(*======================================================================================================================================*)
(*//=============================================================================\\
||  _   _ _  __  _         _                        _   _                      ||
|| | \ | | |/ / / \  _   _| |_ ___  _ __ ___   __ _| |_(_) ___  _ __         ||
|| |  \| | ' / / _ \| | | | __/ _ \| '_ ` _ \ / _` | __| |/ _ \| '_ \        ||
|| | |\  | . \/ ___ \ |_| | || (_) | | | | | | (_| | |_| | (_) | | | |       ||
|| |_| \_|_|\_\_/  \_\__,_|\__\___/|_| |_| |_|\__,_|\__|_|\___/|_| |_|       ||
||                                                                             ||
\\=============================================================================//
SERVOSCHRAUBER - Schraubprozess Schubkastenschiene Nobilia Vorgabe  

Dieser Baustein beschreibt den reinen Schraubprozess, es wird lediglich die 
Motoransteuerung übernommen, alles andere (Pneumatik und Schraubenzuführung) 
kann weiterhin in dem standart Schrauber Baustein stattfinden. Dies sorgt
für eine verbesserte Integration in bereits bestehende Systeme.

Die Gesamte Motoransteuerung findet über die "IQ_SchrauberAchsStruc_InOut" -
Achsstruktur statt, welche zusammen mit dem Baustein aufgerufen und beschrieben
wird. 

Über die "I_stSchraubParam" Struktur werden die Gesamten benötigten Parameter 
an den Schrauber- Baustein übergeben. Diese Struktur kann unverändert
durchgereicht werden.

================================================================================
Vollautomatischer Servoschrauber für Schienen- und Einzelschrauben
mit NC-Achsenanbindung, Drehmoment, Drehwinkel- und Tiefenüberwachung 
================================================================================*)

(*Date          | Version    		| created under     | Author       		| Remark *)
(*====================================================================================================================================================*)
(*23/09/2025   	| 1.00      		| TC3		  		| N.Kersting       	| Neue Isolierte Version *)
(*30/09/2025   	| 1.01      		| TC3		  		| N.Kersting       	| Erste Versuche ohne Motor  *)
(*01/10/2025   	| 1.02      		| TC3		  		| N.Kersting       	| Neue Strukturen Integriert für Prozessdaten etc. *)
(*08/10/2025   	| 1.03      		| TC3		  		| N.Kersting       	| Erste Versuche laufen sehr gut in der Praxis *)
(*09/10/2025   	| 1.04      		| TC3		  		| N.Kersting       	| Merhrere kleine Bugfixe/ Merker wurden nicht Initialisiert... *)
(*09/10/2025   	| 1.05      		| TC3		  		| N.Kersting       	| Drehmomenterhöhung in Schraubfall 1 und 3 nun über Zeit entprellt *)
(*09/10/2025   	| 2.00      		| TC3		  		| N.Kersting       	| Komplette Auswertungsstrategie abgespeckt und anderes konzept, ohne Tiefe zu beachten *)
(*10/10/2025   	| 3.00      		| TC3		  		| N.Kersting       	| Nach Drehmoment Ok wird nun auch die Schraubtiefe in Abhängikeit des Drehwinkels geprüft *)
(*10/10/2025   	| 3.01      		| TC3		  		| N.Kersting       	| Lauffähiger Stand, Auswertung sehr genau, Schraubzeit ca. 500-650ms *)
(*====================================================================================================================================================*)
FUNCTION_BLOCK fb_SKSSchraubNob
VAR_INPUT
	I_bStart			:BOOL;
	I_bFreigabe			:BOOL;
	I_bReset			:BOOL;
	I_bQuittFehler		:BOOL;
	
	I_lrActPosTiefe		:LREAL;
	
	I_stSchraubParam	:ST_SchrauberAblauf_Parameter;	(* Speziefische Parameter für den Schruabprozess *)
	
END_VAR
VAR_OUTPUT
	Q_sState			:STRING;
	Q_bBusy				:BOOL;
	Q_bDone				:BOOL;
	Q_bError			:BOOL;
	Q_nErrorId			:INT;
	Q_bSchrHalt			:BOOL;		(* Motor stoppen *)
	Q_bAxisReset		:BOOL;				(* Achse zurücksetzen *)
	Q_nTorque			:INT := 300;		(* Drehmomentgrenzwert [0.1%] *)
	
	Q_stProzessDaten	:ST_SchrauberAblauf_ProzessDaten;
END_VAR
VAR_IN_OUT
	(* Schraubantrieb Achsstruktur InOut *)
	IQ_SchrauberAchsStruc_InOut		:ST_SchrauberAblauf_AchsStruc;
END_VAR
VAR
	nStep				:INT;
	sStep				:STRING;
	nStepLeerlauf		:INT;
	sStepLeerlauf		:STRING;
	bBusy				: BOOL;
	bDone				: BOOL;
	
	(*========================================================================================================================*)
	(* === PROZESSWERTE === *)
	(*========================================================================================================================*)
	fSchraubTiefeIst				: LREAL;	(* Aktuelle Schraubtiefe [mm] *)
	fDrehmomentIstMittel			: LREAL;	(* Gemitteltes Drehmoment [0.1%] *)
	nTiefeBeimAufsetzen				: LREAL;	(* Tiefe beim ersten Werkstückkontakt *)
	bTiefeBeimAufsetzenOK			: BOOL;		(* Aufsetzen korrekt erkannt *)
	bTiefeOkMem						: BOOL;
	bDrehmomOkMem					: BOOL;
	bDrehwinkelOkMem				: BOOL;
	bTiefeStehtOkMem				: BOOL;
	bSchraubStangeStehtOkMem		: BOOL;
	bDrehwinkelTiefeOkMem			: BOOL;
	nDrehwinkelMem					: LREAL ;
	nTiefErrechnetMem				: LREAL;
	nTiefeAbweichMem				: LREAL;
	nSollDrehmomentErrechnet		: LREAL;	(* Der errechnete Drehmomentwert, Rechnet Drehmoment (Nm) um in Prozessdaten kompatibelen wert für den Antrieb! *)
	bLeerlaufpruefung				: BOOL;
	bDrehmomentErhoehen				: BOOL;			(* Merker Drehmoment erhöhen *)
	bAchsreset						: BOOL;		(* Achsen-Reset intern *)
	lrDrehzahlSollProzent			: LREAL;
	
	(*========================================================================================================================*)
	(* === FEHLERBEHANDLUNG === *)
	(*========================================================================================================================*)
	nFehlerSchrittMerker			: INT;		(* Merker für Fehlerschritt *)
	
	(*========================================================================================================================*)
	(* === Prozessparameter zur Schraubfall auswertung === *)
	(*========================================================================================================================*)
	nAuswertungTiefeMem				: LREAL;	(* Gemerkte Tiefe für Auswertung in Step 60 *)
	nAuswertungPosMem				: LREAL;	(* Gemerkte Position für Auswertung in Step 60 *)
	nMaxDrehwinkel_F3				: LREAL;			
	nDrehwinkelBerechnet			: LREAL; 			(* Der Maximale solldrehwinkel, welcher sich aus der Höhe, wo gestoppt wurde und der Schraubensteigung errechnet *)
	nSchraubFallMerker				: INT;	
	nDrehmomentSkalierVorgabe		: LREAL;
	
	(*========================================================================================================================*)
	(* === Auswertung === *)
	(*========================================================================================================================*)
	fbtimeDiff_Schraub				: fb_timeDiff;
	fbtimeDiff_Komplettt			: fb_timeDiff;
	rTrigPosMem						: r_trig;
	
	(*========================================================================================================================*)
	(* === Zeiten === *)
	(*========================================================================================================================*)
	tonTimeOver						: ton;
	tonDrehmomentErhoehen			: ton;
	
	(*========================================================================================================================*)
	(* === DREHMOMENT-MITTELWERTBILDUNG === *)
	(*========================================================================================================================*)
	arrDrehmomentIst				: ARRAY [0..10] OF LREAL;	(* Ringpuffer für Drehmoment *)
	idx								: INT;		(* Index für Array-Verarbeitung *)
	
	(*========================================================================================================================*)
	(* === Prozesswerte für Analyse === *)
	(*========================================================================================================================*)
	nPD_Tiefe						: LREAL;			(* Prozessdaten - erreichte Tiefe *)
	nPD_Drehmoment					: LREAL;			(* Prozessdaten - erreichtes Drehmoment *)
	nPD_Drehwinkel					: LREAL;			(* Prozessdaten - erreichter Drehwinkel *)
	tPD_Schraubtakt_Komplett		: TIME;				(* Prozessdaten - Zeit für den Kompletten Schraubprozess *)
	tPD_Schraubtakt_Schrauben		: TIME;				(* Prozessdaten - Zeit nur für den Schraubvorgang ohne Zylinder bewegungen etc. *)
	iPD_Schraubfall					: INT;				(* Prozessdaten - Schraubfall *)		
	bPD_SchraubVorgOk				: BOOL;				(* Prozessdaten - Schraubvorgang OK *)
	
	nSollDrehzahl					: INT;
	
	fbtimeDiff_Step45				: fb_timeDiff;
	fbtimeDiff_Step50				: fb_timeDiff;
	fbtimeDiff_Step51				: fb_timeDiff;
	fbtimeDiff_Step55				: fb_timeDiff;
	fbtimeDiff_Step60				: fb_timeDiff;
	fbtimeDiff_Step61				: fb_timeDiff;
	fbtimeDiff_Step62				: fb_timeDiff;
	fbtimeDiff_Step70				: fb_timeDiff;
	fbtimeDiff_Step75				: fb_timeDiff;
	
	stArraySteps					: ARRAY[1..9] OF STRING;
	tGesamtZeit						: TIME;
	sGesamtZeit						: STRING;
	i								: INT;
	rTrigZeitenSchreiben			: R_trig;
	
END_VAR

fSchraubTiefeIst :=	I_lrActPosTiefe;

(* === Hauptablauf === *)
ac_Hauptablauf();

(* === DREHMOMENT-MITTELWERTBILDUNG === *)
m_DrehmomentMittelwert();

(* === SCHRAUBTAKT-ZEITMESSUNG === *)
m_SchraubtaktMessung();

(* === Ausgänge zuweisen === *)
m_Ausgangszuweisung();

ACTION ac_AblaufLeerlaufPruef:
(* ================================================================================ *)
(* LERRLAUF DREHMOMENT PRÜFEN SEQUENZ *)
(* ================================================================================ *)
CASE nStepLeerlauf OF
0: (* === LeerlaufPrüfung/ Erkennung ob Motor Schwergängig ist === *)
	sStepLeerlauf := 'Leerlaufpruefung';
			
	(* Watchdog Positionierfreigabe *)
	tonTimeOver.IN := TRUE;
	tonTimeOver.PT := T#1S;
		
	(* Startdrehzahl setzen *)
	m_DrehzahlVorgabe(
		lrMaxDrehzahl:=  		IQ_SchrauberAchsStruc_InOut.NC_Axis_IN_nParamEilgeschw, 
		lrDrehzahlSollUpm:= 	I_stSchraubParam.nDrehzahlSollEnde, 
		lrDrehzahlVorgabe=> 	lrDrehzahlSollProzent);
			
	(* Drehmoment Vorgabe errechnen *)
	m_DrehmomentVorgabe(
		nSkalierung :=			1,
		nTorque:= 				I_stSchraubParam.nSollmomentLeerlaufPruefung, (* Lerrlaufdrehmoment *) 
		nRatedCurrentMotor:= 	I_stSchraubParam.nNennleistungMotor, 
		nTorqueConstant:= 		I_stSchraubParam.nDrehmomentKonstante, 
		nTorqueLimitation=> 	nSollDrehmomentErrechnet);
		
	Q_nTorque := LREAL_TO_INT(nSollDrehmomentErrechnet);
	
	IF IQ_SchrauberAchsStruc_InOut.NC_Axis_IN_bPTPPosiFreig
	THEN
		tonTimeOver.IN := FALSE;
		
		IQ_SchrauberAchsStruc_InOut.NC_Axis_OUT_nPTPVelo := lrDrehzahlSollProzent;
		IQ_SchrauberAchsStruc_InOut.NC_Axis_OUT_PTPBuffMode := MC_Aborting;
		IQ_SchrauberAchsStruc_InOut.NC_Axis_OUT_bAchsePosStarten := TRUE;	
		nStepLeerlauf := 301;
	ELSIF
		tonTimeOver.Q
	THEN
		tonTimeOver.IN := FALSE;
		nFehlerSchrittMerker := -300;
		nStepLeerlauf := 999;
	END_IF
	
(*================================================================================================================*)
1: (* === LeerlaufPrüfung === *)
	sStepLeerlauf := 'Leerlaufpruefung Auswertung';
	
	(* Watchdog für Leerlauf Prüfung ob Geschwindigkeit mit reduziertem Drehmoment erreicht wurde *)
	(* Watchdog Positionierfreigabe *)
	tonTimeOver.IN := IQ_SchrauberAchsStruc_InOut.NC_Axis_IN_bFaehrtPos;(* Muss noch geguckt werden ob auchh bei Stillstehendem Motor gesetzt wird *)
	tonTimeOver.PT := I_stSchraubParam.tLeerlaufPruefzeit;(* warten damit die Drehzahl erreicht werden kann *)
	
	bLeerlaufpruefung := TRUE;

	(* Wenn 80% der Solldrehzahl erreicht wurde, gilt dies als OK *)
	IF  (((IQ_SchrauberAchsStruc_InOut.NC_Axis_IN_nActVelo / IQ_SchrauberAchsStruc_InOut.NC_Axis_IN_nParamEilgeschw) * 100)
		 >= IQ_SchrauberAchsStruc_InOut.NC_Axis_OUT_nPTPVelo*0.8)
	THEN
		tonTimeOver.IN := FALSE;
		nStepLeerlauf := 999;
	ELSIF
		tonTimeOver.Q
	THEN
		tonTimeOver.IN := FALSE;
		nFehlerSchrittMerker := -301;
		nStepLeerlauf := 999;
	END_IF	

999:;
	
END_CASE
END_ACTION

ACTION ac_Hauptablauf:
(*
================================================================================
HAUPTABLAUF - ZUSTANDSMASCHINE SERVOSCHRAUBER
================================================================================
Zentrale Zustandsmaschine mit deterministischem Ablauf.
Alle Schritte sind eindeutig nummeriert und kommentiert.
Watchdog-Timer überwachen kritische Phasen.
================================================================================
*)

tonTimeOver();

(*=== HAUPTZUSTANDSMASCHINE === *)
IF NOT I_bReset 
THEN
	CASE nStep OF
(*================================================================================================================*)	
	(* ================================================================================ *)
	(* INITIALISIERUNG UND BEREITSCHAFT *)
	(* ================================================================================ *)
(*================================================================================================================*)
	0: (* === INITIALISIERUNG === *)
		sStep := 'Initialisierung';
		bDone := FALSE;
		
		(* Drehmoment Vorgabe errechnen *)
		m_DrehmomentVorgabe(
			nSkalierung :=			I_stSchraubParam.nDrehmomentSkalierVorgabe,
			nTorque:= 				I_stSchraubParam.nDrehmomentSoll * I_stSchraubParam.nDrehmomentSkalierVorgabe, (* Drehmoment erst Senken um Überdrehen zu verhinder *) 
			nRatedCurrentMotor:= 	I_stSchraubParam.nNennleistungMotor, 
			nTorqueConstant:= 		I_stSchraubParam.nDrehmomentKonstante, 
			nTorqueLimitation=> 	nSollDrehmomentErrechnet);
			
		Q_nTorque := LREAL_TO_INT(nSollDrehmomentErrechnet); 
		
		IF I_bFreigabe
		THEN
			nStep := 10;
		END_IF
		
(*================================================================================================================*)
	10: (* === BEREITSCHAFT === *)
		sStep := 'Bereitschaft';
		tonTimeOver.IN := FALSE;
		tonDrehmomentErhoehen.IN := FALSE;
		
		(* Drehmoment Vorgabe errechnen *)
		m_DrehmomentVorgabe(
			nSkalierung :=			I_stSchraubParam.nDrehmomentSkalierVorgabe,
			nTorque:= 				I_stSchraubParam.nDrehmomentSoll * I_stSchraubParam.nDrehmomentSkalierVorgabe, (* Drehmoment erst Senken um Überdrehen zu verhinder *) 
			nRatedCurrentMotor:= 	I_stSchraubParam.nNennleistungMotor, 
			nTorqueConstant:= 		I_stSchraubParam.nDrehmomentKonstante, 
			nTorqueLimitation=> 	nSollDrehmomentErrechnet);
			
		Q_nTorque := LREAL_TO_INT(nSollDrehmomentErrechnet); 
		bBusy							:= TRUE;
		
		IF I_bStart
			AND Q_nTorque <>0
		THEN
			(* Prozessdaten auf 0 setzen *)
			nPD_Tiefe						:= 0;			(* Prozessdaten - erreichte Tiefe *)
			nPD_Drehmoment					:= 0;			(* Prozessdaten - erreichtes Drehmoment *)
			nPD_Drehwinkel					:= 0;			(* Prozessdaten - erreichter Drehwinkel *)
			tPD_Schraubtakt_Komplett		:= T#0S;		(* Prozessdaten - Zeit für den Kompletten Schraubprozess *)
			tPD_Schraubtakt_Schrauben		:= T#0S;		(* Prozessdaten - Zeit nur für den Schraubvorgang ohne Zylinder bewegungen etc. *)
			iPD_Schraubfall					:= 0;			(* Prozessdaten - Schraubfall *)		
			bPD_SchraubVorgOk				:= FALSE;		(* Prozessdaten - Schraubvorgang OK *)
			nDrehwinkelMem     				:= 0;
			bDrehmomOkMem					:= FALSE;
			bDrehwinkelOkMem				:= FALSE;
			bTiefeOkMem						:= FALSE;
			bTiefeStehtOkMem				:= FALSE;
			bDrehmomentErhoehen				:= FALSE;
			bSchraubStangeStehtOkMem		:= FALSE;
			bDrehwinkelTiefeOkMem			:= FALSE;
			nTiefeAbweichMem				:= 0;
			nFehlerSchrittMerker			:= 0;
			nSchraubFallMerker				:= 0;
			nTiefErrechnetMem				:= 0;
			nStep := 45;
		END_IF
		
(*================================================================================================================*)
	45: (* === ANLAUFPHASE - LANGSAME DREHZAHL === *)
		sStep := 'Anlaufphase_Langsam';
					
		(* Watchdog für Anlaufphase *)
		tonTimeOver.IN := TRUE;
		tonTimeOver.PT := T#5S;
	
		(* Startdrehzahl setzen *)
		m_DrehzahlVorgabe(
			lrMaxDrehzahl:=  		IQ_SchrauberAchsStruc_InOut.NC_Axis_IN_nParamEilgeschw, 
			lrDrehzahlSollUpm:= 	I_stSchraubParam.nDrehzahlSollAnfang, 
			lrDrehzahlVorgabe=> 	lrDrehzahlSollProzent);
			
		IQ_SchrauberAchsStruc_InOut.NC_Axis_OUT_nPTPVelo := lrDrehzahlSollProzent;
		IQ_SchrauberAchsStruc_InOut.NC_Axis_OUT_PTPBuffMode := MC_Aborting;
		IQ_SchrauberAchsStruc_InOut.NC_Axis_OUT_bAchsePosStarten := I_bFreigabe;
		
		(* Prüfung ob 80% der Sollgeschwindigkeit erreicht *)
		IF	IQ_SchrauberAchsStruc_InOut.NC_Axis_IN_bFaehrtPos 
		    AND (((IQ_SchrauberAchsStruc_InOut.NC_Axis_IN_nActVelo / IQ_SchrauberAchsStruc_InOut.NC_Axis_IN_nParamEilgeschw) * 100)
			     >= IQ_SchrauberAchsStruc_InOut.NC_Axis_OUT_nPTPVelo * 0.8)
		THEN
			
			IQ_SchrauberAchsStruc_InOut.NC_Axis_OUT_bAchsePosStarten := FALSE;
			tonTimeOver.IN := FALSE;
			nStep := 50;	(* -> Hauptschraubphase *)
			
		ELSIF tonTimeOver.Q 
		THEN
			(* Timeout - Geschwindigkeit nicht erreicht *)
			tonTimeOver.IN := FALSE;
			nStep := 70;	(* -> Motor stoppen *)
			nFehlerSchrittMerker := -45;	(* Fehlercode merken *)
		END_IF
		
(*================================================================================================================*)
	50: (* === HAUPTSCHRAUBPHASE - GESCHWINDIGKEIT AUFBAUEN === *)
		sStep := 'Hauptschraubphase_Beschleunigen';
		
		(* Watchdog für Beschleunigungsphase *)
		tonTimeOver.IN := TRUE;
		tonTimeOver.PT := T#3S;
			
		IQ_SchrauberAchsStruc_InOut.NC_Axis_OUT_bAchsePosStarten := I_bFreigabe;
		
		(* Prozessdaten Tiefe Schreiben *)
		nPD_Tiefe:=	fSchraubTiefeIst;
		
		(* Startdrehzahl setzen *)
		m_DrehzahlVorgabe(
			lrMaxDrehzahl:=  		IQ_SchrauberAchsStruc_InOut.NC_Axis_IN_nParamEilgeschw, 
			lrDrehzahlSollUpm:= 	I_stSchraubParam.nDrehzahlSoll, 
			lrDrehzahlVorgabe=> 	lrDrehzahlSollProzent);
			
		(* Umschaltung auf Solldrehzahl basierend auf Schraubtiefe *)
		IF I_bStart 
			AND fSchraubTiefeIst < I_stSchraubParam.nTiefeSollDrehzahl 
		THEN
			(* Vollschraubung *)
			tonTimeOver.IN := FALSE;
			IQ_SchrauberAchsStruc_InOut.NC_Axis_OUT_bAchsePosStarten := FALSE;
			IQ_SchrauberAchsStruc_InOut.NC_Axis_OUT_nPTPVelo := lrDrehzahlSollProzent;
			IQ_SchrauberAchsStruc_InOut.NC_Axis_OUT_PTPBuffMode := MC_BlendingNext;
			IQ_SchrauberAchsStruc_InOut.NC_Axis_OUT_bAchsePosStarten := I_bFreigabe;
			nStep := 51;	(* -> Drehzahlabsenkung *)
		ELSIF 
			tonTimeOver.Q 
		THEN
			(* Timeout - Solltiefe für Drehzahlumschaltung nicht erreicht *)
			tonTimeOver.IN := FALSE;
			nStep := 70;	(* -> Motor stoppen *)
			nFehlerSchrittMerker := -50;	(* Fehlercode merken *)
		END_IF
		
(*================================================================================================================*)
	51: (* === Warten Auf Velo Verringert === *)
		sStep := 'Hauptschraubphase_Drehzahl verringern';	
		
		(* Watchdog für Beschleunigungsphase *)
		tonTimeOver.IN := TRUE;
		tonTimeOver.PT := I_stSchraubParam.tZeitdSchraubTakt;
			
		(* Startdrehzahl setzen *)
		m_DrehzahlVorgabe(
			lrMaxDrehzahl:=  		IQ_SchrauberAchsStruc_InOut.NC_Axis_IN_nParamEilgeschw, 
			lrDrehzahlSollUpm:= 	I_stSchraubParam.nDrehzahlSollEnde, 
			lrDrehzahlVorgabe=> 	lrDrehzahlSollProzent);
		
		(* Aufruf Drehmoment Prüfen *)
		m_DrehmomentPruefung(
			nDrehmomentSoll:= 		I_stSchraubParam.nDrehmomentSoll, 
			bDrehmomentOk=> 		bDrehmomOkMem);
	
		IF fSchraubTiefeIst < I_stSchraubParam.nTiefeLangsamDrehzahl
			OR bDrehmomOkMem	(* Nun auch schon vorher gucken ob das Drehmoment nicht doch schon kommt um Drehzahl zu Reduzieren *)
		THEN
			(* Vollschraubung *)
			IQ_SchrauberAchsStruc_InOut.NC_Axis_OUT_bAchsePosStarten := I_bFreigabe;
			IQ_SchrauberAchsStruc_InOut.NC_Axis_OUT_nPTPVelo := lrDrehzahlSollProzent  ;	
			IQ_SchrauberAchsStruc_InOut.NC_Axis_OUT_PTPBuffMode := MC_BlendingNext;
			IQ_SchrauberAchsStruc_InOut.NC_Axis_OUT_bAchsePosStarten := I_bFreigabe;
		
			(* Warten, dass 80% der iSt Drehzahl kleiner ist als die Soll Drehzahl  *)
			IF IQ_SchrauberAchsStruc_InOut.NC_Axis_IN_bFaehrtPos 
				AND (((IQ_SchrauberAchsStruc_InOut.NC_Axis_IN_nActVelo*0.8 / IQ_SchrauberAchsStruc_InOut.NC_Axis_IN_nParamEilgeschw) * 100)
					 <= IQ_SchrauberAchsStruc_InOut.NC_Axis_OUT_nPTPVelo)	
			THEN
				tonTimeOver.IN := FALSE;
				nStep := 55;	
			END_IF
			
		ELSIF
			tonTimeOver.Q
		THEN			
			tonTimeOver.IN := FALSE;
			nFehlerSchrittMerker := -51;	(* -> Timeout Kein Drehmoment und keine Tiefe *) (* Fehlercode merken *)
			nStep := 70;	
		END_IF
		
(*================================================================================================================*)
	55: (* === Schraubfallauswertung === *)
		sStep := 'Schraubfall Auswertung';
		
		(* Watchdog für Auswertung Schraubfall *)
		tonTimeOver.IN := TRUE;
		tonTimeOver.PT := I_stSchraubParam.tSchraubfallAuswertung;
			
		IQ_SchrauberAchsStruc_InOut.NC_Axis_OUT_bAchsePosStarten := I_bFreigabe;
		
		(* Startdrehzahl setzen *)
		m_DrehzahlVorgabe(
			lrMaxDrehzahl:=  		IQ_SchrauberAchsStruc_InOut.NC_Axis_IN_nParamEilgeschw, 
			lrDrehzahlSollUpm:= 	I_stSchraubParam.nDrehzahlSollEnde, 
			lrDrehzahlVorgabe=> 	lrDrehzahlSollProzent);
		
		(* Tiefenprüfung *)
		IF I_bStart
		THEN
			m_TiefenPruefung(
				nSolltiefeMin:= 	I_stSchraubParam.nMinimalSchraubtiefe, 
				nSolltiefeMax:= 	I_stSchraubParam.nSchraubtiefeSoll, 
				nToleranz:= 		0,	 
				nActTiefe:= 		fSchraubTiefeIst, 
				bTiefeOk=> 			bTiefeOkMem);
		END_IF
		
		(* Aufruf Drehmoment Prüfen *)
		m_DrehmomentPruefung(
			nDrehmomentSoll:= 		I_stSchraubParam.nDrehmomentSoll, 
			bDrehmomentOk=> 		bDrehmomOkMem);
					
		IF bDrehmomOkMem
		THEN
			tonTimeOver.IN := FALSE;
			IQ_SchrauberAchsStruc_InOut.NC_Axis_OUT_nPTPVelo := lrDrehzahlSollProzent ;	
			nSchraubFallMerker :=	1;
			nStep := 60;
		ELSIF
			 tonTimeOver.Q 
		THEN							
			tonTimeOver.IN := FALSE;
			nFehlerSchrittMerker := -55;	(* -> Timeout Drehmoment erreichen *) (* Fehlercode merken *)
			nStep := 70;	
		END_IF
		
(*================================================================================================================*)
	60: (* === Warten Auf Velo Verringert === *)
		sStep := 'Schraubfall Auswertung';	
		
		(* Watchdog für Schraubvorgang *)
		tonTimeOver.IN := TRUE;
		tonTimeOver.PT :=  I_stSchraubParam.tZeitdSchraubTakt;
		
		(* Warten, dass 80% der iSt Drehzahl kleiner ist als die Soll Drehzahl  *)
		IF IQ_SchrauberAchsStruc_InOut.NC_Axis_IN_bFaehrtPos 
		    AND (((IQ_SchrauberAchsStruc_InOut.NC_Axis_IN_nActVelo*0.8 / IQ_SchrauberAchsStruc_InOut.NC_Axis_IN_nParamEilgeschw) * 100)
			     <= IQ_SchrauberAchsStruc_InOut.NC_Axis_OUT_nPTPVelo)
		THEN
			nAuswertungPosMem := IQ_SchrauberAchsStruc_InOut.NC_Axis_IN_nActPos; (* Position Merken, wo Drehmoment erreicht wurde *)	
			nAuswertungTiefeMem :=	fSchraubTiefeIst; (* Tiefe Merken, wo Drehmoment erreicht wurde *)
					
			nStep := 61;	
		ELSIF
			tonTimeOver.Q
		THEN			
			tonTimeOver.IN := FALSE;
			nFehlerSchrittMerker := -60;	(* -> Timeout Drehzahl Absenken *) (* Fehlercode merken *)
			nStep := 70;	
		END_IF
		
(*================================================================================================================*)			
	61:	(* === Schraubfall === *) 
		ac_Schraubfall();	
		
(*================================================================================================================*)			
	62:	(* === Tiefenänderung prüfen === *) 
		ac_TiefenAuswertung();
		
(*================================================================================================================*)			
(*	63:	(* === Schraubfall 3 === *) 
		ac_Schraubfall3();		*)
		
(*================================================================================================================*)
	70: (* === MOTOR STOPPEN === *)
		sStep := 'Motor_Stoppen';
		Q_nTorque := 0;
		
		(* Watchdog für Stoppvorgang *)
		tonTimeOver.IN := TRUE;
		tonTimeOver.PT :=  T#100MS;
				
		(* Achse stoppen *)
		IQ_SchrauberAchsStruc_InOut.NC_Axis_OUT_bAchsePosStoppen := TRUE;
		
		(* Warten auf Stillstand *)
		IF tonTimeOver.Q 
		   OR IQ_SchrauberAchsStruc_InOut.NC_Axis_IN_bInPos
		THEN
			tonTimeOver.IN := FALSE;
			IQ_SchrauberAchsStruc_InOut.NC_Axis_OUT_bAchsePosStoppen := FALSE;
			IQ_SchrauberAchsStruc_InOut.NC_Axis_OUT_bAchsePosStarten := FALSE;
			nStep := 75;	(* -> Stillstand abwarten *)
		END_IF
		
(*================================================================================================================*)
	75: (* === STILLSTAND ABWARTEN === *)
		sStep := 'Stillstand_Abwarten';
		
		(* Watchdog für Stillstand *)
		tonTimeOver.IN := TRUE;
		tonTimeOver.PT :=  T#2S;
		
		(* Warten auf Motorstillstand *)
		IF tonTimeOver.Q
			OR IQ_SchrauberAchsStruc_InOut.NC_Axis_IN_bInStillstand
		THEN
			bAchsreset := TRUE;
			tonTimeOver.IN := FALSE;
			
			nStep := 80;
		END_IF

(*================================================================================================================*)
	80: (* === AUSWERTUNG FEHLERSCHRITTMERKER === *)
		sStep := 'Fehlerschritt auswerten';
		
		(* Fehler auswerten *)
		IF nFehlerSchrittMerker <> 0
		THEN
			nStep := nFehlerSchrittMerker;
		ELSE
			bPD_SchraubVorgOk := TRUE;
			nStep := 100;
		END_IF
				
(*================================================================================================================*)
	100: (* === VORGANG ERFOLGREICH BEENDET === *)
		sStep := 'Vorgang_OK';
		
		bBusy := FALSE;
		bDone := TRUE;
		
		(* Warten auf Freigabe für nächsten Zyklus *)
		IF NOT I_bStart 
		THEN
			bLeerlaufpruefung := FALSE;
			Q_nTorque := 300;	
			IQ_SchrauberAchsStruc_InOut.NC_Axis_OUT_bSteuerwortBit1	:= FALSE;
			IQ_SchrauberAchsStruc_InOut.NC_Axis_OUT_bAchsePosStarten := FALSE;
			nStep := 0;	(* -> Zurück zur Bereitschaft *)
		END_IF
		
(*================================================================================================================*)
	(* ================================================================================ *)
	(* LERRLAUF DREHMOMENT PRÜFEN SEQUENZ *)
	(* ================================================================================ *)
	300: sStep := sStepLeerlauf;
				
		ac_AblaufLeerlaufPruef();
		
		IF nStepLeerlauf = 999
		THEN
			nStepLeerlauf :=0;
			nStep := 70;
		END_IF
		
(*================================================================================================================*)
	(* ================================================================================ *)
	(* FEHLERBEHANDLUNG *)
	(* ================================================================================ *)
		
(*================================================================================================================*)
	-45: (* === FEHLER: LANGSAME GESCHWINDIGKEIT === *)
		sStep := 'FEHLER: Langsame Geschwindigkeit wird nicht erreicht';
		Q_nErrorId := -45;
		
		IF I_bQuittFehler 
		THEN
			nStep := 100;	(* -> Beenden *)
		END_IF
		
(*================================================================================================================*)
	-50: (* === FEHLER: SCHRAUBTIEFE FÜR SOLLDREHZAHL === *)
		sStep := 'FEHLER: Schraubtiefe für Solldrehzahl wird nicht erreicht';
		Q_nErrorId := -50;
		
		IF I_bQuittFehler 
		THEN
			nStep := 100;	(* -> Beenden *)
		END_IF
		
(*================================================================================================================*)
	-55: (* === FEHLER:  === *)
		sStep := 'FEHLER: Timeout Drehmoment- Auswertung';
		Q_nErrorId := -55;
		
		IF I_bQuittFehler 
		THEN
			nStep := 100;	(* -> Beenden *)
		END_IF
		
(*================================================================================================================*)		
	-60: (* === FEHLER:  === *)
		sStep := 'FEHLER: Timeout abbremsen';
		Q_nErrorId := -60;
		
		IF I_bQuittFehler 
		THEN
			nStep := 100;	(* -> Beenden *)
		END_IF
		
(*================================================================================================================*)
(* === FEHLER: Schraubfall 1  === *)		
(*================================================================================================================*)
	-61: 
		sStep := 'FEHLER: Schraubfall 1 Undefiniert- Timeout';
		Q_nErrorId := -61;
		
		IF I_bQuittFehler 
		THEN
			nStep := 100;	(* -> Beenden *)
		END_IF
		
(*================================================================================================================*)
	-1261: 
		sStep := 'FEHLER: Schraubfall 1 Drehwinkel Überschritten';
		Q_nErrorId := -1261;
		
		IF I_bQuittFehler 
		THEN
			nStep := 100;	(* -> Beenden *)
		END_IF	
		
(*================================================================================================================*)
	-62: 
		sStep := 'FEHLER: Tiefe hat sich geändert obwohl Drehmoment OK';
		Q_nErrorId := -62;
		
		IF I_bQuittFehler 
		THEN
			nStep := 100;	(* -> Beenden *)
		END_IF
		
(*================================================================================================================*)
	-301: (* === FEHLER: Leerlaufprüfung === *)
		sStep := 'FEHLER: Leerlauf Drehzahl nicht erreicht, Schwergang?';
		Q_nErrorId := -301;
		
		IF I_bQuittFehler 
		THEN
			nStep := 100;	(* -> Beenden *)
		END_IF
		
(*================================================================================================================*)
	-300: (* === FEHLER: Leerlaufprüfung === *)
		sStep := 'FEHLER: Leerlaufprüfung keine Freigabe zum Positionieren';
		Q_nErrorId := -300;
		
		IF I_bQuittFehler 
		THEN
			nStep := 100;	(* -> Beenden *)
		END_IF
		
	END_CASE
	
ELSE
	(* === RESET AKTIV === *)
	nStep := 0;
END_IF

(*========================================================*)
(* Prozessdaten Merker schreiben *)
(*========================================================*)
IF (nStep >= 55)
	AND (nStep <= 70)
THEN
	(* Prozessdaten Drehwinkel Schreiben *)
	IF nDrehwinkelMem> nPD_Drehwinkel
	THEN
		nPD_Drehwinkel :=	nDrehwinkelMem;
	END_IF
	(* Prozessdaten Tiefe Schreiben *)
	IF fSchraubTiefeIst < nPD_Tiefe
	THEN
		nPD_Tiefe:=	fSchraubTiefeIst;
	END_IF
	(* Prozessdaten Drehmoment Schreiben *)
	IF fDrehmomentIstMittel >nPD_Drehmoment
	THEN
		nPD_Drehmoment :=	fDrehmomentIstMittel;
	END_IF
	
	iPD_Schraubfall :=	nSchraubFallMerker;
END_IF

(*========================================================*)
(* Prozessdaten Struktur schreiben *)
(*========================================================*)
Q_stProzessDaten.nPD_Drehmoment				:=	nPD_Drehmoment;
Q_stProzessDaten.nPD_Drehwinkel				:=	nPD_Drehwinkel;
Q_stProzessDaten.nPD_Tiefe					:=	nPD_Tiefe;
Q_stProzessDaten.tPD_Schraubtakt_Komplett	:=	tPD_Schraubtakt_Komplett;
Q_stProzessDaten.tPD_Schraubtakt_Schrauben	:=	tPD_Schraubtakt_Schrauben;
Q_stProzessDaten.iPD_Schraubfall			:=	iPD_Schraubfall;
Q_stProzessDaten.bPD_SchraubVorgOk			:=	bPD_SchraubVorgOk;
Q_stProzessDaten.bPD_DrehmomOk				:=	bDrehmomOkMem;
Q_stProzessDaten.bPD_DrehwinkelOk			:=	bDrehwinkelOkMem;
Q_stProzessDaten.bPD_TiefeOk				:=	bTiefeOkMem;
END_ACTION

ACTION ac_Schraubfall:
(*================================================================================================================*)
(* === Drehwinkelprüfung&  Drehmoment Prüfung === *)
(*
Fall 1 – Moment OK, Tiefe nicht OK
- Ausgangslage: Verbindung zieht, Tiefe fehlt noch.
- Ziel: Tiefer eindrehen, ohne Überdrehen.
- Vorgehen:
  - Weiterdrehen mit großer Winkelreserve.
  - Reserve aus fehlender Tiefe + Schraubensteigung berechnet,
    plus kleiner Nachziehwinkel.
- Stop: Tiefe erreicht innerhalb Reserve → Stopp.
- Eskalation: Tiefe kommt nicht → Moment moderat erhöhen.
- Abbruch: Timeout oder Winkelobergrenze überschritten.*)
(*================================================================================================================*)

sStep := 'Schraubvorgang Auswertung Drehwinkel und Drehmoment';

(* Watchdog für Schraubvorgang *)
tonTimeOver.IN := 	TRUE;
tonTimeOver.PT :=	I_stSchraubParam.tZeitdSchraubfallTimeout;

Q_nTorque := LREAL_TO_INT(nSollDrehmomentErrechnet );	(* Drehmoment wieder Setzen damit der Motor weiter drehen kann *)

(* Aufruf Drehwinkel Prüfen *)
m_DrehwinkelPruefung(
	nPosAct:= 			IQ_SchrauberAchsStruc_InOut.NC_Axis_IN_nActPos, 
	nPosMem:= 			nAuswertungPosMem, 
	nPosSoll:= 			I_stSchraubParam.nSollDrehwinkelNachDrehmomOK, (* mindest Drehwinkel nach Drehmoment ok *)
	nMaxDrehwinkel :=	I_stSchraubParam.nMaxDrehwinkelNachDrehmOk, (* Maximal Drehwinkel nach Drehmoment ok *)
	bWinkelOk=> 		bDrehwinkelOkMem,
	nWinkelAct=>		nDrehwinkelMem);

(* Aufruf Drehmoment Prüfen *)
m_DrehmomentPruefung(
	nDrehmomentSoll:= 		I_stSchraubParam.nDrehmomentSoll, 
	bDrehmomentOk=> 		bDrehmomOkMem);

(* Aufruf Schrauberstange auf Stillstand Prüfen *)	
m_StillstandPruef(
	nIstDrehzahl:= 		IQ_SchrauberAchsStruc_InOut.NC_Axis_IN_nActVelo, 
	nMinDrehzahl:= 		ABS(IQ_SchrauberAchsStruc_InOut.NC_Axis_IN_nParamEilgeschw * 0.01), (* 1% der Bezugsgeschwindigkeit *)
	bSteht=> 			bSchraubStangeStehtOkMem);
	
IF NOT tonTimeOver.Q
THEN
	IF 	ABS(nDrehwinkelMem) <I_stSchraubParam.nMaxDrehwinkelNachDrehmOk	(* Nur abfragen ob nicht überdreht *)
		AND bSchraubStangeStehtOkMem (* Schrauberstange dreht sich nicht mehr *) 
		AND bDrehmomOkMem
	THEN 	
		tonTimeOver.IN := 	FALSE;
		Q_nTorque := 0;
		nStep := 62;	(* -> Motor stoppen *)
	ELSIF
		ABS(nDrehwinkelMem) >(I_stSchraubParam.nMaxDrehwinkelNachDrehmOk)
	THEN
		(* Wenn Drehwinkel Überschritten-> Direkt Anhalten *)
		tonTimeOver.IN := 	FALSE;
		nStep := 70;	(* -> Motor stoppen *)
		nFehlerSchrittMerker := -1261;	(* Fehlercode merken Drehwinkel Überschritten Fall 1*)			
	END_IF
ELSE
	nFehlerSchrittMerker := -61;
	tonTimeOver.IN := 	FALSE;
	nStep := 70;	(* -> Motor stoppen *)
END_IF
END_ACTION

ACTION ac_TiefenAuswertung:
(* Watchdog für Tiefenänderung *)
tonTimeOver.IN := TRUE;
tonTimeOver.PT :=  T#100MS;

m_TiefenAenderung(
	nTiefeStreckeIst:= 		ABS(fSchraubTiefeIst) -ABS(nAuswertungTiefeMem), 
	nDrehwinkelIst:= 		nDrehwinkelMem, 
	nSteigungSchraube:= 	I_stSchraubParam.nHoeheSchraubenDrehung, 
	nAbweichung:= 			25, 
	nTiefeErrechnet=> 		nTiefErrechnetMem, 
	nProzentAbweichung=>	nTiefeAbweichMem,
	bTiefeSteht=> 			bTiefeStehtOkMem);
 
IF bTiefeStehtOkMem
THEN
	tonTimeOver.IN := 	FALSE;
	Q_nTorque := 0;
	nStep := 70;	(* -> Motor stoppen *)
ELSIF
	tonTimeOver.Q
THEN
	(* Wenn bTiefeStehtOkMem bedeutet dies, dass der Schraubenkopf noch nicht anliegt, 
		weiterer Umgang muss noch Folgen, aber erst mal Fehler*)
	tonTimeOver.IN := FALSE;
	nFehlerSchrittMerker := -62;	(* -> Tiefe hat sich geändert Logik muss noch folgen, aber erst mal Fehler *) (* Fehlercode merken *)
	nStep := 70;
END_IF
END_ACTION

ACTION ac99_Doku:
(*
## 1. Überblick / Zweck
Der Baustein `fb_SKSSchraubNob` kapselt den **reinen servo‑motorischen Schraubprozess** (Drehzahl-, Drehmoment-, Winkel- und Tiefenführung) und lässt alle peripheren Funktionen (z. B. Pneumatik, Schraubenzuführung) im bestehenden Standard-Schrauberbaustein. Dadurch kann der Motor-Schraubkern in bestehende Anlagen integriert werden, ohne tiefgreifende Umbauten in der Peripherie vornehmen zu müssen.  
Unterstützt werden:
- Drehmomentüberwachung  
- Drehwinkelberechnung / -begrenzung  
- Tiefenerfassung (Position entspricht Einschraubtiefe)  
- Klassifizierung des Verlaufs in definierte Schraubfälle  
- Zeit- und Qualitätsauswertung  

## 2. Integration in einen vorhandenen Schrauberablauf
Einbettung erfolgt typischerweise so:
1. Bestehender Ablauf (PnP / Handlingslogik) positioniert Werkzeug, versorgt Schraube, setzt ggf. Pneumatik.
2. Achsstruktur (IN/OUT) wird an den Baustein übergeben (standardisierte Servoantriebs-Schnittstelle).
3. Parametrierstruktur (Schraubparameter) wird 1:1 durchgereicht (keine Aufsplittung nötig).
4. Start-/Freigabe-/Reset-/Quittiersignale kommen aus übergeordneter Ablaufsteuerung.
5. Prozessdaten (Tiefe, Drehmoment, Winkel, Dauer, Klassifikation) werden nach Abschluss zurückgemeldet und können für Trace, Qualität oder MES erfasst werden.
6. Fehler- oder Schraubfall-Ergebnis kann direkt in nachfolgende Entscheider (OK/NOK/Sortierung) einfließen.

Vorteile:
- Plug-in für bestehenden Schrauber-Ablauf .
- Leichte Austauschbarkeit oder parallele Variantenentwicklung.
- Geringeres Risiko bei Änderungen (nur Kernlogik betroffen).
- Einheitliche Achsschnittstelle fördert Wiederverwendung.

## 3. Architektur & Zustandslogik (technischer Überblick)
Der Baustein verwendet eine deterministische Zustandsmaschine (nummerierte Schritte). Kernphasen:
1. Initialisierung / Bereitschaft
2. Anlauf mit reduzierter Drehzahl
3. Übergang auf Hauptdrehzahl
4. Drehzahlreduktion vor Auswertung
5. Schraubfall-Erkennung (Entscheidung: welcher Verlauf liegt vor?)
6. Feinschraubphase je nach Schraubfall (1, 2 oder 3)
7. Bremsen / Stillsetzen
8. Ergebnis- und Fehlerauswertung
9. Rückkehr in Bereitschaft

Ergänzend: eigene Sequenz zur Leerlauf-/Schwergangprüfung mit separater Unter-Zustandsmaschine.

## 4. Schraubfälle (Klassifikation des Verlaufs)
Die Klassifikation beruht auf der Relation zwischen erreichten Zielgrößen (Tiefe, Drehmoment) zum Zeitpunkt der Auswertung:

| Schraubfall | Auslöser (Situation) | Zielstrategie | Typische Maßnahmen | Abbruchkriterien |
|-------------|----------------------|---------------|--------------------|------------------|
| 1 | Drehmoment erreicht, Tiefe noch nicht | Weiter eindringen ohne Überdrehen | Winkelreserve aus fehlender Tiefe + Nachziehreserve, ggf. Drehmoment moderat erhöhen | Timeout, Winkelgrenze überschritten |
| 2 | Tiefe erreicht, Drehmoment noch nicht | Vorspannung sauber aufbauen | Begrenztes Nachdrehen in kleinem Winkel-Fenster | Timeout (Moment fehlt), Fenster überschritten |
| 3 | Weder Tiefe noch Moment erreicht | Beides sicher erreichen | Zunächst größere Winkel-/Tiefenreserve, dann Übergang wie Fall 1 bzw. 2 | Timeout, Winkelobergrenze |
| Leerlaufprüfung | Vor dem eigentlichen Prozess: Antrieb läuft „frei“ | Erkennen von Schwergang / Blockade | Prüfen ob Geschwindigkeit mit reduziertem Moment erreicht wird | Timeout oder zu niedrige Drehzahl |

Zusammenfassung:
- Fall 1: Verbindung zieht früh (Moment da), Schraube steht noch sichtbar über Oberfläche.
- Fall 2: Schraube liegt bündig (Tiefe da), aber Vorspannung fehlt noch.
- Fall 3: „Träger Verlauf“ – weder Tiefe noch Moment früh erreicht, daher weiter beobachten und adaptiv reagieren.
- Leerlaufprüfung: Schutzmechanismus / Frühdiagnose.

## 5. Ablaufbeschreibung 
1. Der Baustein wartet, bis die übergeordnete Steuerung signalisiert, dass alles bereit ist (Werkzeug positioniert, Schraube vorhanden, Sicherheitsfreigaben aktiv).
2. Beim Start setzt er interne Messgrößen (z. B. Zähler und Qualitätsmerker) zurück.
3. Der Schraubvorgang beginnt langsam, um ein ruckfreies Ansetzen sicherzustellen und frühe Auffälligkeiten (Blockade, verkantete Schraube) zu erkennen.
4. Erhöht sich die Einschraubtiefe wie erwartet, wird beschleunigt, um Zeit zu sparen.
5. Kurz vor einer vorgesehenen Übergangszone wird wieder auf eine niedrigere Geschwindigkeit reduziert, um kontrolliert in den sensiblen Bereich (Finalisierung) einzufahren.
6. Nun vergleicht das System: Ist bereits die benötigte Tiefe erreicht? Ist das gewünschte Drehmoment erzielt? Aus dieser Kombination erkennt es, welcher Verlauf vorliegt.
7. Je nach Verlauf wendet es ein passendes Feinkonzept an:
   - Schraubfall 1: Nur Tiefe fehlt → etwas weiter eindrehen, ohne zu fest anzuziehen.
   - Schraubfall 2: Nur Drehmoment fehlt → gezielte Nachdrehung, begrenzt im Winkel.
   - Schraubfall 3: Beides fehlt → weitere kontrollierte Bewegung, mit eventueller Anpassung.
8. Währenddessen wird laufend das Drehmoment gemittelt um Ausreißer zu filtern.
9. Erreichen alle Zielgrößen gültige Werte (Tiefe im Fenster, Drehmoment ausreichend, Winkel nicht zu groß), wird der Antrieb gestoppt.
10. Der Prozess wird protokolliert: Zeitbedarf, erreichte Tiefe, maximales Drehmoment, gedrehter Winkel und Klassifikation.
11. Bei Unregelmäßigkeiten (z. B. Zeit überschritten, Winkel zu groß) markiert das System den Vorgang als fehlerhaft und wartet auf eine Quittierung.
12. Nach Freigabe für den nächsten Zyklus kehrt der Baustein in die Ausgangsbereitschaft zurück.


## 6. Prozessdaten (Ergebnis- / Qualitätsdaten)
| Name (Ausgabe) | Bedeutung | Einheit | Hinweise |
|----------------|----------|---------|----------|
| nPD_Tiefe | Erreichte minimale Einschraubtiefe (negativer Weg oder mm je nach Bezug) | mm | Wird während der aktiven Phase aktualisiert (kleinster Wert, falls Tiefe Richtung Werkstück negativ zählt) |
| nPD_Drehmoment | Höchstes gemitteltes Drehmoment im Prozess | % (0.1%-Skalierung) oder intern skaliert | Basierend auf Mittelwertbildung zur Glättung |
| nPD_Drehwinkel | Größter errechneter/erfasster Drehwinkel (Differenz seit Auswertungspunkt) | Grad / Umdrehungsäquivalent | Berechnet aus Achsposition und Steigung |
| tPD_Schraubtakt_Komplett | Gesamtzeit von Start bis Abschluss/Fehler | Zeit | Für Taktoptimierung |
| tPD_Schraubtakt_Schrauben | Reine Schraubzeit (ohne z. B. Zylinderwege) | Zeit | Differenziert Ursachen von Verzögerungen |
| iPD_Schraubfall | Klassifizierter Schraubfall (1–3) | Zahl | 0 vor Auswertung |
| bPD_SchraubVorgOk | Gesamt-OK-Flag des Vorgangs | BOOL | FALSE bei Fehler oder Abbruch |
| bPD_DrehmomOk | Soll-Drehmoment erreicht | BOOL | Teilkriterium Qualität |
| bPD_DrehwinkelOk | Nachdreh-/Winkelkriterium erfüllt | BOOL | Verhindert Überdrehen |
| bPD_TiefeOk | Tiefe innerhalb Toleranzfenster | BOOL | Oberflächenbündigkeit / Setzpunkt |

## 7. Parameterbeschreibung (Eingabestruktur)
(Hinweis: Nicht alle Parameter der Struktur waren vollständig sichtbar. Liste basiert auf den im Code referenzierten Feldern.)

| Parameter | Bedeutung / Funktion | Einheit / Bereich | Wirkung / Bemerkungen |
|-----------|----------------------|-------------------|-----------------------|
| nDrehzahlSollAnfang | Anfangsdrehzahl für Schon-Anlauf | U/min | Reduziert Risiko von Verkanten |
| nDrehzahlSoll | Hauptdrehzahl (Schnellphase) | U/min | Produktivgeschwindigkeit |
| nDrehzahlSollEnde | Reduzierte Drehzahl in Feinschraubphase | U/min | Feinfühliges Erreichen der Ziele |
| nTiefeSollDrehzahl | Einschraubtiefe, ab der auf Hauptdrehzahl hochgeschaltet wird | mm | Umschaltkriterium Beschleunigung |
| nTiefeLangsamDrehzahl | Einschraubtiefe, ab der wieder verlangsamt wird | mm | Vorbereitung Feinauswertung |
| nMinimalSchraubtiefe | Untere Toleranzgrenze für Tiefe | mm | Qualitätsfenster |
| nSchraubtiefeSoll | Zieltiefe | mm | Nennwert Tiefe |
| nDrehmomentSoll | Ziel-Drehmoment | Skaliert / % / Nm-Äquivalent | Referenz für Freigabekriterium |
| nDrehmomentSkalierVorgabe | Globaler Skalierungsfaktor | Faktor | Multipliziert Ziel-Moment (z. B. Softstart) |
| nDrehmomentSkalVerringern | Temporäre Reduktion für Brems-/Übergangsphase | Faktor | Vor Auswertung wird Moment gesenkt |
| nDrehmomentErhoehung | Zusatzmoment bei Fall 1 / 3 wenn Tiefe „hängt“ | Skaliert | Adaptive Nachregelung |
| nSollmomentLeerlaufPruefung | Momentbegrenzung in Leerlaufprüfung | % / skaliert | Erkennung Schwergang ohne Schäden |
| tLeerlaufPruefzeit | Prüfzeitfenster Leerlauf | Zeit | Timeout-Kriterium |
| tZeitdSchraubTakt | Allgemeines Zeitlimit für Teilphasen / Nachziehfenster | Zeit | Wiederverwendetes Watchdog-Intervall |
| tSchraubfallAuswertung | Spezifisches Zeitfenster für Klassifikation | Zeit | Verhindert endloses Abwarten |
| nHoeheSchraubenDrehung | Steigung (Tiefe pro Umdrehung oder pro Segment) | mm/U | Grundlage für Winkelberechnung |
| nSollDrehwinkelNachTiefeOK | Mindestnachdrehwinkel nach Tiefeerfüllung | Grad | Sicherstellung Setzvorgang |
| nDrehwinkelNachziehen_F1 | Zusatz-Winkelreserve bei Fall 1 | Grad | Verhindert Untervorspannung |
| nMaxDrehwinkelNachTiefeOk_F1 | Sicherheitslimit Fall 1 | Grad | Abbruch bei Überdrehung |
| nMaxDrehwinkelNachTiefeOk_F2 | Sicherheitslimit Fall 2 | Grad | Engeres Fenster |
| (vermutet) nMaxDrehwinkel_F3 | Limit für Fall 3 (im Code angelegt) | Grad | Analog Fall 1/2 (nicht komplett sichtbar) |
| nNennleistungMotor | Referenz Motorstrom / Bemessung | A / % | Für Berechnung Drehmomentgrenze |
| nDrehmomentKonstante | Umrechnungsfaktor (Strom→Moment) | Nm/A | Erforderlich für physikalische Skalierung |
*)
END_ACTION

METHOD m_Ausgangszuweisung : BOOL
VAR_INPUT
END_VAR
(*
================================================================================
AUSGANGSZUWEISUNG
================================================================================
Zentrale Zuweisung aller Ausgangssignale mit Sicherheitsverriegelung
durch Schutzbereich und Reset-Zustand
================================================================================
*)

// === HAUPTSTATUS-AUSGÄNGE ===
Q_bBusy		:= bBusy;				(* Beschäftigt wenn nicht in Bereitschaft *)

Q_bDone		:= bDone;		(* Fertig bei Schritt 100 *)

// === ACHSEN-STEUERUNG ===
Q_bAxisReset := bAchsreset;

// === DIAGNOSE-AUSGÄNGE ===
Q_sState	:= sStep(*CONCAT(INT_TO_STRING(nStep), CONCAT(' - ', sStep))*);

Q_bSchrHalt := (nStep = 70);

(* Fehler allgemein *)
Q_bError	:= nStep<0;
END_METHOD

METHOD m_DrehmomentMittelwert : BOOL
VAR_INPUT
END_VAR
(*
================================================================================
DREHMOMENT-MITTELWERTBILDUNG
================================================================================
Berechnet den gleitenden Mittelwert des Drehmoments über 10 Werte
zur Vermeidung von Fehlauslösungen durch kurze Spitzen.
================================================================================
*)
// === MITTELWERTBILDUNG NUR WÄHREND DREHMOMENTPRÜFUNG ===
IF (nStep >= 51 
	AND nStep <= 70) 
	OR nStep =301
THEN
	m_DrehmomentRechnung(
		nTorqueActValue:= 		INT_TO_LREAL(IQ_SchrauberAchsStruc_InOut.NC_Axis_IN_nActTorque), 
		nRatedCurrentMotor:=	I_stSchraubParam.nNennleistungMotor , 	
		nTorqueConstant:= 		I_stSchraubParam.nDrehmomentKonstante, 
		nActTorqueCalc=> 		arrDrehmomentIst[0]);
	
	// Array nach rechts verschieben (Ringpuffer)
	FOR idx := 10 TO 1 BY -1 DO
		arrDrehmomentIst[idx] := arrDrehmomentIst[idx-1];
	END_FOR
	
	// Mittelwert über alle 10 Werte berechnen
	fDrehmomentIstMittel := (arrDrehmomentIst[1] 
						   + arrDrehmomentIst[2] 
						   + arrDrehmomentIst[3] 
						   + arrDrehmomentIst[4] 
						   + arrDrehmomentIst[5] 
						   + arrDrehmomentIst[6] 
						   + arrDrehmomentIst[7] 
						   + arrDrehmomentIst[8] 
						   + arrDrehmomentIst[9] 
						   + arrDrehmomentIst[10]) / 10;
ELSE
	fDrehmomentIstMittel := 0;
END_IF
END_METHOD

METHOD m_DrehmomentPruefung : BOOL
VAR_INPUT
	nDrehmomentSoll		:LREAL;				
END_VAR
VAR_OUTPUT
	bDrehmomentOk		:BOOL;
END_VAR
(*
================================================================================
DrehmomentPruefung
================================================================================
Berechnet den gleitenden Mittelwert des Drehmoments über 10 Werte
zur Vermeidung von Fehlauslösungen durch kurze Spitzen.
================================================================================
*)
IF fDrehmomentIstMittel >= 
	nDrehmomentSoll
THEN
	bDrehmomentOk := TRUE;	(* -> Drehmoment erreicht *)
ELSE
	bDrehmomentOk := FALSE;	
END_IF
END_METHOD

METHOD m_DrehmomentRechnung : BOOL
VAR_INPUT
	
	
	nTorqueActValue		:LREAL;	
	
	nRatedCurrentMotor	:LREAL;	(*0x8011:12	*)
	nTorqueConstant		:LREAL;	(*0x8011:16	*)
END_VAR
VAR_OUTPUT
	nActTorqueCalc		:LREAL;
END_VAR
(*Achtung dies aus der Original Beckhoff Doku:

Anzeige des aktuellen Drehmomentwertes
Der Wert wird in 1000stel vom rated current (0x8011:12
[} 151]) angegeben
Formel für Index 0x8010:54 [} 148] = 0 :
M = ((Torque actual value / 1000) x (rated current /
√2)) x torque constant (0x8011:16 [} 151])
Formel für Index 0x8010:54 [} 148] = 1 :
M = ((Torque actual value / 1000) x rated current)) x
torque constant (0x8011:16 [} 151])*)
nActTorqueCalc:=	
(((nTorqueActValue/1000) * (nRatedCurrentMotor / 1.4142))* nTorqueConstant);		(* Wurzel ziehen am besten einmalig bei Startup *)
END_METHOD

METHOD m_DrehmomentVorgabe : BOOL
VAR_INPUT
	nSkalierung			:LREAL;
	nTorque				:LREAL;		(* Eingang Soll Drehmoment in Nm	*)
	
	nRatedCurrentMotor	:LREAL;	(*0x8011:12	*)
	nTorqueConstant		:LREAL;	(*0x8011:16	*)
END_VAR
VAR_OUTPUT
	nTorqueLimitation	:LREAL;
END_VAR
(*Achtung dies aus der Original Beckhoff Doku:

Anzeige des aktuellen Drehmomentwertes
Der Wert wird in 1000stel vom rated current (0x8011:12
[} 151]) angegeben
Formel für Index 0x8010:54 [} 148] = 0 :
M = ((Torque actual value / 1000) x (rated current /
√2)) x torque constant (0x8011:16 [} 151])
Formel für Index 0x8010:54 [} 148] = 1 :
M = ((Torque actual value / 1000) x rated current)) x
torque constant (0x8011:16 [} 151])*)
nTorqueLimitation := ((nTorque / nTorqueConstant) / (nRatedCurrentMotor / 1.4142)) * 1000 *nSkalierung;
END_METHOD

METHOD m_DrehwinkelPruefung : BOOL
VAR_INPUT
	nPosAct		:LREAL;	(* Aktuelle Position  *)
	nPosMem		:LREAL;	(* Gespeicherte Position *)
	nPosSoll	:LREAL; (* Soll Drehwinkel *)
	nMaxDrehwinkel	:LREAL;
	
END_VAR
VAR_OUTPUT
	bWinkelOk			:BOOL;
	nWinkelAct	:LREAL;
END_VAR
VAR
	
END_VAR
nWinkelAct :=	nPosAct-nPosMem;

bWinkelOk :=	nWinkelAct > nPosSoll 
				AND nWinkelAct < nMaxDrehwinkel;
END_METHOD

METHOD m_DrehzahlVorgabe 
VAR_INPUT
	lrMaxDrehzahl		:LREAL;		(* Drhezahl Eilgeschwindigkeit in Grad/ sec *)
	lrDrehzahlSollUpm	:LREAL;		(* Drehzahl Soll in Upm *)
END_VAR
VAR
	lrDrehzahlMem		:LREAL;
	
END_VAR
VAR_OUTPUT
	lrDrehzahlVorgabe	:LREAL;			(* Soll Drehzahl in % von 100 % *)
END_VAR
lrDrehzahlMem := lrMaxDrehzahl /360 *60;

IF lrDrehzahlMem <> 0
THEN
	lrDrehzahlVorgabe :=	lrDrehzahlSollUpm / lrDrehzahlMem *100;
END_IF
END_METHOD

METHOD m_SchraubtaktMessung : BOOL
VAR_INPUT
END_VAR
(*
================================================================================
SCHRAUBTAKT-ZEITMESSUNG
================================================================================
Misst die Schraubzeit für Diagnose und Optimierung.
Die Zeitmessung erfolgt während der aktiven Schraubphase.
================================================================================
*)
(* Komplett wird nicht verwendet, da ausgelagert in dem Übergeordneten Schrauberbaustein *)
(*fbtimeDiff_Komplettt(
	bStart:= 		(nStep =10),	 
	bStop:= 		(nStep =100), 
	bReset:= 		(nStep =10),
	tDiffTime=> 	tPD_Schraubtakt_Komplett);*)
	
tPD_Schraubtakt_Komplett := T#0MS;

(* Zeitmessung Schruabvorgang *)
fbtimeDiff_Schraub(
	bStart:= 		(nStep =45),	 
	bStop:= 		(nStep =80), 
	bReset:= 		(nStep =10),
	tDiffTime=> 	tPD_Schraubtakt_Schrauben);

	
fbtimeDiff_Step45(
	bStart:= 			nStep =45, 
	bStop:= 			nStep <>45, 
	bReset:= 			nStep = 10);

fbtimeDiff_Step50(
	bStart:= 			nStep =50, 
	bStop:= 			nStep <>50, 
	bReset:= 			nStep = 10);
	
fbtimeDiff_Step51(
	bStart:= 			nStep =51, 
	bStop:= 			nStep <>51, 
	bReset:= 			nStep = 10);
	
fbtimeDiff_Step55(
	bStart:= 			nStep =55, 
	bStop:= 			nStep <>55, 
	bReset:= 			nStep = 10);
	
fbtimeDiff_Step60(
	bStart:= 			nStep =60, 
	bStop:= 			nStep <>60, 
	bReset:= 			nStep = 10);
	
fbtimeDiff_Step45(
	bStart:= 			nStep =45, 
	bStop:= 			nStep <>45, 
	bReset:= 			nStep = 10);
	
fbtimeDiff_Step61(
	bStart:= 			nStep =61, 
	bStop:= 			nStep <>61, 
	bReset:= 			nStep = 10);
	
fbtimeDiff_Step62(
	bStart:= 			nStep =62, 
	bStop:= 			nStep <>62, 
	bReset:= 			nStep = 10);

fbtimeDiff_Step70(
	bStart:= 			nStep =70, 
	bStop:= 			nStep <>70, 
	bReset:= 			nStep = 10);

fbtimeDiff_Step75(
	bStart:= 			nStep =75, 
	bStop:= 			nStep <>75, 
	bReset:= 			nStep = 10);	
	
(* Zeiten Schreiben *)
rTrigZeitenSchreiben(CLK:= (nStep =100));

IF rTrigZeitenSchreiben.Q
THEN
	stArraySteps[1] :=	CONCAT('Step_45_LangsamEin: ', INT_TO_STRING(TIME_TO_INT(fbtimeDiff_Step45.tDiffTime )));
	stArraySteps[2] :=	CONCAT('Step_50_Beschleunigen auf SollDrehzahl: ', INT_TO_STRING(TIME_TO_INT(fbtimeDiff_Step50.tDiffTime )));
	stArraySteps[3] :=	CONCAT('Step_51_Umschaltung Langsame Drehzahl: ', INT_TO_STRING(TIME_TO_INT(fbtimeDiff_Step51.tDiffTime )));
	stArraySteps[4] :=	CONCAT('Step_55_Warte auf Drehmoment: ', INT_TO_STRING(TIME_TO_INT(fbtimeDiff_Step55.tDiffTime )));
	stArraySteps[5] :=	CONCAT('Step_60_Warte auf Drehzahl verringert: ', INT_TO_STRING(TIME_TO_INT(fbtimeDiff_Step60.tDiffTime )));
	stArraySteps[6] :=	CONCAT('Step_61_Auswertung Drehmoment und Drehwinkel: ', INT_TO_STRING(TIME_TO_INT(fbtimeDiff_Step61.tDiffTime )));
	stArraySteps[7] :=	CONCAT('Step_62_Auswertung Tiefenänderung: ', INT_TO_STRING(TIME_TO_INT(fbtimeDiff_Step62.tDiffTime )));
	stArraySteps[8] :=	CONCAT('Step_70_Motor anhalten: ', INT_TO_STRING(TIME_TO_INT(fbtimeDiff_Step70.tDiffTime )));
	stArraySteps[9] :=	CONCAT('Step_75_Warte auf Motor Steht: ', INT_TO_STRING(TIME_TO_INT(fbtimeDiff_Step75.tDiffTime )));
	
	tGesamtZeit:=	fbtimeDiff_Step45.tDiffTime
					+	fbtimeDiff_Step50.tDiffTime
					+	fbtimeDiff_Step51.tDiffTime
					+	fbtimeDiff_Step55.tDiffTime
					+	fbtimeDiff_Step60.tDiffTime
					+	fbtimeDiff_Step61.tDiffTime
					+	fbtimeDiff_Step62.tDiffTime
					+	fbtimeDiff_Step70.tDiffTime
					+	fbtimeDiff_Step75.tDiffTime;
					
	sGesamtZeit :=		CONCAT('GesamtZeit: ', INT_TO_STRING(TIME_TO_INT(tGesamtZeit )));
END_IF
END_METHOD

METHOD m_StillstandPruef 
VAR_INPUT
	nIstDrehzahl	:LREAL;
	nMinDrehzahl	:LREAL;
END_VAR
VAR_OUTPUT
	bSteht			:BOOL;
END_VAR




IF ABS(nIstDrehzahl) < ABS(nMinDrehzahl) 
THEN
	bSteht := TRUE;
ELSE
	bSteht := FALSE;
END_IF
END_METHOD

METHOD m_TiefenAenderung
VAR_INPUT
	nTiefeStreckeIst				:LREAL;
	nDrehwinkelIst					:LREAL;
	nSteigungSchraube				:LREAL := 1.6;	(* Tiefe pro umdrehung *)
	nAbweichung						:LREAL := 25;	(* in Prozent *)
END_VAR
VAR_OUTPUT
	nProzentAbweichung 				:LREAL;	(* Nur zu Diagnosezwecken *)
	nTiefeErrechnet					:LREAL;	(* Nur zu Diagnosezwecken *)
	bTiefeSteht						:BOOL;
END_VAR
VAR
	nDelta             : LREAL;
END_VAR

IF nSteigungSchraube  > 0
	AND nAbweichung > 0
THEN
	nTiefeErrechnet :=	ABS(nDrehwinkelIst /360* nSteigungSchraube);
	
	nDelta := ABS(nTiefeErrechnet - nTiefeStreckeIst);
	
    IF nTiefeStreckeIst <> 0.0 THEN
        nProzentAbweichung := nDelta / ABS(nTiefeStreckeIst) * 100.0;
    ELSE
        nProzentAbweichung := 0.0;
    END_IF

    IF nProzentAbweichung >= nAbweichung THEN
        bTiefeSteht := TRUE;
    ELSE
        bTiefeSteht := FALSE;
    END_IF
	
ELSE
    bTiefeSteht := FALSE;
    nTiefeErrechnet := 0.0;
END_IF
END_METHOD

METHOD m_TiefenPruefung : BOOL
VAR_INPUT
	nSolltiefeMin	:LREAL;
	nSolltiefeMax	:LREAL;
	nToleranz	:LREAL;
	nActTiefe	:LREAL;
END_VAR
VAR_OUTPUT
	bTiefeOk	:BOOL;
END_VAR
// Prüfung der Aufsetztiefe
IF F_Inbetween(
	I_fActualValue := nActTiefe,
	I_fMinimalValue := nSolltiefeMin - nToleranz,		(* Sollaufsetztiefe ± Toleranz *)
	I_fMaximalValue := nSolltiefeMax + nToleranz) 
THEN
	bTiefeOk := TRUE;
ELSE
	bTiefeOk := FALSE;
END_IF
END_METHOD

END_FUNCTION_BLOCK

(* stored: Version 1.1.0.1, ProductVersion 3.1.4024.15
   POU fb_SKSSchraubNob: Id {7264520c-c401-4547-9877-f980c7765746}, SpecialFunc None
   Folder Ablauf: Id {fafa4d6d-6f22-46f3-bf08-cf1d510a3348}
   Folder Ausgang: Id {6aba5681-4e5c-480a-99f0-c6a63017ffef}
   Folder Auswertung: Id {6546e813-580a-4c40-8d8a-37f1e1c6b5fe}
   Folder Diagnose: Id {30f33323-bedf-4681-9716-d32c8fe17ccb}
   Folder Drehmoment: Id {4f4c9446-1ae7-4f1c-abfe-f801565df70b}
   Folder Pruefung: Id {85b2db60-3bc3-4c45-ab1d-146f31338f7e}
   Folder Rechner: Id {a1e596fa-1c68-4ed0-91bf-d850752cd9d3}
   Action ac_AblaufLeerlaufPruef: Id {5b9e4dbf-dd31-408e-8211-c2f059162955}
   Action ac_Hauptablauf: Id {a7beba71-c765-4242-9292-6d5fa44c1eae}
   Action ac_Schraubfall: Id {5c67398b-963c-4b49-9885-21994fb5412b}
   Action ac_TiefenAuswertung: Id {270db67a-4949-4c92-912d-219e1e9ec108}
   Action ac99_Doku: Id {4b2e4e7e-3f57-4148-b830-7a58c66f56ce}
   Method m_Ausgangszuweisung: Id {74c01e09-c989-4b6c-9bb0-bfec5129497b}
   Method m_DrehmomentMittelwert: Id {77f39372-f3e1-4000-849a-5801781248c7}
   Method m_DrehmomentPruefung: Id {b15c2951-703a-4b2e-94f4-6e1a127b2d05}
   Method m_DrehmomentRechnung: Id {1bbcef17-e04b-4f43-82fa-b98e6a4d6400}
   Method m_DrehmomentVorgabe: Id {334d5570-7cec-4c2d-8d0e-4201a4c66404}
   Method m_DrehwinkelPruefung: Id {f7872583-c9f4-4570-9dc0-fe102e0e693a}
   Method m_DrehzahlVorgabe: Id {d8955cdf-71ce-4acf-ba19-552d62bfa9a7}
   Method m_SchraubtaktMessung: Id {0bd72a6b-78b6-4b56-acc0-b6d291daa095}
   Method m_StillstandPruef: Id {78e76abc-3570-46f3-b0f9-5b0c754e0a13}
   Method m_TiefenAenderung: Id {4331bc38-e923-4719-8891-74280cf938a9}
   Method m_TiefenPruefung: Id {a103558d-0397-404b-aa38-f8b16ef7498c} *)
